{attribute 'qualified_only'}
VAR_GLOBAL

	fb_mcp		: FB_mcp;
	
	status	: MachineStatus := MachineStatus.STOPPED;
	
	iAng_air AT%I* :INT;
	aiFlow AT%I* :INT;


	PackTags					: ST_PackMLv30;					//PackTags

	nVisuProductCommand			: DINT;							//Products to produce

	bButtonProductionReq		: BOOL;							//TRUE when a mode change to PRODUCTION is requested
	stChangeIntoProduction		: ST_ChangeIntoProduction;		//Result of command box "Change to Production requested"

	aUnitInfo					: ARRAY [1..12] OF ST_UnitInfo;	//Array includes the states and modes of machineunits	
	aCaption					: ARRAY [1..12] OF STRING := ['F1','F2','F3','F4','F5','F6','F7','F8','F9','F10','F11','F12'];
	aKeyPressed					: ARRAY [1..12] OF BOOL;		
	
	alarm_empty		: ST_Alarm;
	alarm_temp		: ST_Alarm;
	str				: STRING;
	pml_adminAlarm	: PML_AdminAlarm;		
	

	fb_sample	: FB_Sample;
	
END_VAR
VAR_GLOBAL CONSTANT
	iAlarm_max	:INT	:= 19;
	rAir_setting	: REAL	:=0.4;
END_VAR

(* stored: Version 1.1.0.1, ProductVersion 3.1.4024.12
   GVL GVL: Id {467ff484-abc3-43b3-a376-da9ea4486a4c} *)
